FUNCTION TryConvert_WORD_TO_LREAL : BOOL
VAR_INPUT
	in : WORD;
	out : REFERENCE TO LREAL;
END_VAR

out := WORD_TO_LREAL(in);
TryConvert_WORD_TO_LREAL := TRUE;

END_FUNCTION

(* stored: Version 1.1.0.1, ProductVersion 3.1.4024.12
   POU TryConvert_WORD_TO_LREAL: Id {b3d26687-8bc0-4930-a1e0-32ebfc11de4c}, SpecialFunc None *)
